(* Logix 5000 project; controller Hose_HP_Test_Rig_V1 vendor 1 type 14 code 149 rev 32.11; software revision 32.00; part 7 of 10 *)
(* tags used below, declared in another part *)
   GOTO_FAIL_BIN_STN1 : DINT;
   GOTO_FAULT_BIN_STN3 : DINT;
   PASS_COUNTER_STN1 : COUNTER;
   PASS_COUNTER_STN2 : COUNTER;
   PASS_COUNTER_STN3 : COUNTER;
   PASS_COUNTER_STN4 : COUNTER;
   ACT_PR_STN1 : REAL;
   ACT_PR_STN2 : REAL;
   ACT_PR_STN3 : REAL;
   ACT_PR_STN4 : REAL;
   AUTO_DOOR_OPEN_ON : BOOL;
   AUTO_DOOR_OPEN_ON_STN3 : BOOL;
   AUTO_TEST_ON_STN1 : BOOL;
   AUTO_TEST_ON_STN2 : BOOL;
   AUTO_TEST_ON_STN3 : BOOL;
   AUTO_TEST_ON_STN4 : BOOL;
   BOTTOM_CLAMP_AUTO_STN1 : BOOL;
   BOTTOM_CLAMP_AUTO_STN3 : BOOL;
   BOTTOM_CLAMP_C : REAL;
   BOTTOM_CLAMP_PR : REAL;
   BOTTOM_CLAMP_PR_SEL : BOOL;
   BOTTOM_CLAMP_PR_SEL_SET : BOOL;
   BOTTOM_CLAMP_PR_SEL_SOL : ALIAS FOR REM:O.Data[1].7;
   BOTTOM_CLAMP_SET_STN1 : BOOL;
   BOTTOM_CLAMP_SET_STN3 : BOOL;
   BOTTOM_CLAMP_SOL_STN1 : ALIAS FOR Local:1:O.Data.4;
   BOTTOM_CLAMP_SOL_STN3 : ALIAS FOR Local:3:O.Data.4;
   BOTTOM_CLAMP_X : REAL;
   BOTTOM_CLAMP_X1 : REAL;
   BOTTOM_CLAMP_X2 : REAL;
   BOTTOM_CLAMP_Y1 : REAL;
   BOTTOM_CLAMP_Y2 : REAL;
   BOTTOM_DECLAMP_AUTO_STN1 : BOOL;
   BOTTOM_DECLAMP_AUTO_STN3 : BOOL;
   BOTTOM_DECLAMP_SET_STN1 : BOOL;
   BOTTOM_DECLAMP_SET_STN3 : BOOL;
   BOTTOM_DECLAMP_SOL_STN1 : ALIAS FOR REM:O.Data[0].3;
   BOTTOM_DECLAMP_SOL_STN3 : ALIAS FOR REM:O.Data[0].7;
   BOTTOM_PR_SCL : SCP;
   BUZZER_STN1 : ALIAS FOR Local:3:O.Data.20;
   BUZZER_STN3 : ALIAS FOR Local:3:O.Data.29;
   CONS_FAIL_COUNT_STN1 : DINT;
   CONS_FAIL_COUNT_STN2 : DINT;
   CONS_FAIL_COUNT_STN3 : DINT;
   CONS_FAIL_COUNT_STN4 : DINT;
   CONS_FAIL_COUNTER_STN1 : COUNTER;
   CONS_FAIL_COUNTER_STN2 : COUNTER;
   CONS_FAIL_COUNTER_STN3 : COUNTER;
   CONS_FAIL_COUNTER_STN4 : COUNTER;
   CONSTRICTION_FILL_VAL_STN1 : BOOL;
   CONSTRICTION_FILL_VAL_STN3 : BOOL;
   CONSTRICTION_VALVE_SET_STN1 : BOOL;
   CONSTRICTION_VALVE_SET_STN3 : BOOL;
   DICH2_1_32 : DINT;
   DOOR_CLOSE_ABORT_STN1 : BOOL;
   DOOR_CLOSE_ABORT_STN3 : BOOL;
   DOOR_CLOSE_AUTO_STN1 : BOOL;
   DOOR_CLOSE_AUTO_STN3 : BOOL;
   DOOR_CLOSE_SET_STN1 : BOOL;
   DOOR_CLOSE_SET_STN3 : BOOL;
   DOOR_CLOSE_SOL_STN1 : ALIAS FOR Local:1:O.Data.2;
   DOOR_CLOSE_SOL_STN3 : ALIAS FOR Local:3:O.Data.2;
   DOOR_OPEN_SET_STN1 : BOOL;
   DOOR_OPEN_SET_STN3 : BOOL;
   DOOR_OPEN_SOL_STN1 : ALIAS FOR Local:1:O.Data.1;
   DOOR_OPEN_SOL_STN3 : ALIAS FOR Local:3:O.Data.1;
   EMG_FAULTED_STN1 : BOOL;
   EMG_FAULTED_STN3 : BOOL;
   EXHAUST_SET_STN1 : BOOL;
   EXHAUST_SET_STN3 : BOOL;
   EXHAUST_VALVE_STN1 : ALIAS FOR Local:1:O.Data.7;
   EXHAUST_VALVE_STN3 : ALIAS FOR Local:3:O.Data.7;
   EXHS_VAL_HP_ON_STN1 : BOOL;
   EXHS_VAL_HP_ON_STN3 : BOOL;
   EXHS_VAL_ON_STN1 : BOOL;
   EXHS_VAL_ON_STN3 : BOOL;
   FAIL_COUNT_RETEST : DINT;
   FAIL_COUNT_RETEST_STN2 : DINT;
   FAIL_COUNT_STN1 : DINT;
   FAIL_COUNT_STN2 : DINT;
   FAIL_COUNT_STN3 : DINT;
   FAIL_COUNT_STN4 : DINT;
   FAIL_COUNTER_RETEST : COUNTER;
   FAIL_COUNTER_RETEST_STN2 : COUNTER;
   FAIL_COUNTER_STN1 : COUNTER;
   FAIL_COUNTER_STN2 : COUNTER;
   FAIL_COUNTER_STN3 : COUNTER;
   FAIL_COUNTER_STN4 : COUNTER;
   FAILED_STN1 : BOOL;
   FAILED_STN3 : BOOL;
   FAULT_COUNT_STN1 : DINT;
   FAULT_COUNT_STN2 : DINT;
   FAULT_COUNT_STN3 : DINT;
   FAULT_COUNT_STN4 : DINT;
   FAULT_COUNTER_STN1 : COUNTER;
   FAULT_COUNTER_STN2 : COUNTER;
   FAULT_COUNTER_STN3 : COUNTER;
   FAULT_COUNTER_STN4 : COUNTER;
   FAULT_LAMP_STN1 : ALIAS FOR Local:3:O.Data.19;
   FAULT_LAMP_STN3 : ALIAS FOR Local:3:O.Data.28;
   FAULTED_STN1 : BOOL;
   FAULTED_STN3 : BOOL;
   FINAL_PR_BOTTOM_CLAMP : BOOL;
   FINAL_PR_STN1 : BOOL;
   FINAL_PR_STN2 : BOOL;
   FINAL_PR_STN3 : BOOL;
   FINAL_PR_STN4 : BOOL;
   FINAL_PR_TOP_CLAMP : BOOL;
   GOTO_FAIL_BIN_STN3 : DINT;
   GOTO_FAULT_BIN_STN1 : DINT;
   HIDE_MAIN_MENU : BOOL;
   HP_FILL_VALVE_SET_STN1 : BOOL;
   HP_FILL_VALVE_SET_STN3 : BOOL;
   HP_FILL_VALVE_STN1 : ALIAS FOR Local:1:O.Data.8;
   HP_FILL_VALVE_STN3 : ALIAS FOR Local:3:O.Data.8;
   INITIAL_PR_BOTTOM_CLAMP : BOOL;
   INITIAL_PR_STN1 : BOOL;
   INITIAL_PR_STN2 : BOOL;
   INITIAL_PR_STN3 : BOOL;
   INITIAL_PR_STN4 : BOOL;
   INITIAL_PR_TOP_CLAMP : BOOL;
   INPUT_1_16 : INT;
   MASTER_PR : REAL;
   MASTER_PR_CONS : REAL;
   MASTER_PR_SCL : SCP;
   MSB_EIP_1_16 : INT;
   PASS_COUNT_RETEST : DINT;
   PASS_COUNT_RETEST_STN2 : DINT;
   PASS_COUNT_STN1 : DINT;
   PASS_COUNT_STN2 : DINT;
   PASS_COUNT_STN3 : DINT;
   PASS_COUNT_STN4 : DINT;
   PASS_COUNTER_RETEST : COUNTER;
   PASS_COUNTER_RETEST_STN2 : COUNTER;
   PASS_LAMP_STN1 : ALIAS FOR Local:3:O.Data.18;
   PASS_LAMP_STN3 : ALIAS FOR Local:3:O.Data.27;
   PASSED_STN1 : BOOL;
   PASSED_STN3 : BOOL;
   PR_C_MASTER : REAL;
   PR_C_STAMP : REAL;
   PR_C_STN1 : REAL;
   PR_C_STN2 : REAL;
   PR_C_STN3 : REAL;
   PR_C_STN4 : REAL;
   PR_C_WORK : REAL;
   PR_DIFF_CALB_ACT : REAL;
   PR_SCL_STN1 : SCP;
   PR_SCL_STN2 : SCP;
   PR_SCL_STN3 : SCP;
   PR_SCL_STN4 : SCP;
   PR_X1_MASTER : REAL;
   PR_X1_STAMP : REAL;
   PR_X1_STN1 : REAL;
   PR_X1_STN2 : REAL;
   PR_X1_STN3 : REAL;
   PR_X1_STN4 : REAL;
   PR_X1_WORK : REAL;
   PR_X2_MASTER : REAL;
   PR_X2_STAMP : REAL;
   PR_X2_STN1 : REAL;
   PR_X2_STN2 : REAL;
   PR_X2_STN3 : REAL;
   PR_X2_STN4 : REAL;
   PR_X2_WORK : REAL;
   PR_X_MASTER : REAL;
   PR_X_STAMP : REAL;
   PR_X_STN1 : REAL;
   PR_X_STN2 : REAL;
   PR_X_STN3 : REAL;
   PR_X_STN4 : REAL;
   PR_X_WORK : REAL;
   PR_Y1_MASTER : REAL;
   PR_Y1_STAMP : REAL;
   PR_Y1_STN1 : REAL;
   PR_Y1_STN2 : REAL;
   PR_Y1_STN3 : REAL;
   PR_Y1_STN4 : REAL;
   PR_Y1_WORK : REAL;
   PR_Y2_MASTER : REAL;
   PR_Y2_STAMP : REAL;
   PR_Y2_STN1 : REAL;
   PR_Y2_STN2 : REAL;
   PR_Y2_STN3 : REAL;
   PR_Y2_STN4 : REAL;
   PR_Y2_WORK : REAL;
   RESET_COUNT_RETEST : BOOL;
   RESET_COUNT_RETEST_STN2 : BOOL;
   RESET_COUNT_STN1 : BOOL;
   RESET_COUNT_STN2 : BOOL;
   RESET_COUNT_STN3 : BOOL;
   RESET_COUNT_STN4 : BOOL;
   RST_BOTTOM_DECLAMP_STN1 : BOOL;
   RST_BOTTOM_DECLAMP_STN3 : BOOL;
   RST_DOOR_OPEN_ON : BOOL;
   RST_DOOR_OPEN_ON_STN3 : BOOL;
   RST_TOP_DECLAMP_AUTO_STN1 : BOOL;
   RST_TOP_DECLAMP_AUTO_STN3 : BOOL;
   STAMP_ON_STN1 : BOOL;
   STAMP_ON_STN3 : BOOL;
   STAMP_PR : REAL;
   STAMP_PR_SCL : SCP;
   STAMP_SOL_STN1 : ALIAS FOR Local:1:O.Data.5;
   STAMP_SOL_STN3 : ALIAS FOR Local:3:O.Data.5;
   STS : DINT;
   TEST_LAMP_STN1 : ALIAS FOR Local:3:O.Data.17;
   TEST_LAMP_STN3 : ALIAS FOR Local:3:O.Data.26;
   TEST_SOL_STN1 : ALIAS FOR Local:1:O.Data.6;
   TEST_SOL_STN3 : ALIAS FOR Local:3:O.Data.6;
   TEST_VAL_ON_STN1 : BOOL;
   TEST_VAL_ON_STN3 : BOOL;
   TOP_CLAMP_AUTO_STN1 : BOOL;
   TOP_CLAMP_AUTO_STN3 : BOOL;
   TOP_CLAMP_C : REAL;
   TOP_CLAMP_PR : REAL;
   TOP_CLAMP_PR_SEL : BOOL;
   TOP_CLAMP_PR_SEL_SET : BOOL;
   TOP_CLAMP_PR_SEL_SOL : ALIAS FOR REM:O.Data[1].6;
   TOP_CLAMP_SET_STN1 : BOOL;
   TOP_CLAMP_SET_STN3 : BOOL;
   TOP_CLAMP_SOL_STN1 : ALIAS FOR Local:1:O.Data.3;
   TOP_CLAMP_SOL_STN3 : ALIAS FOR Local:3:O.Data.3;
   TOP_CLAMP_X : REAL;
   TOP_CLAMP_X1 : REAL;
   TOP_CLAMP_X2 : REAL;
   TOP_CLAMP_Y1 : REAL;
   TOP_CLAMP_Y2 : REAL;
   TOP_DECLAMP_AUTO_STN1 : BOOL;
   TOP_DECLAMP_AUTO_STN3 : BOOL;
   TOP_DECLAMP_SET_STN1 : BOOL;
   TOP_DECLAMP_SET_STN3 : BOOL;
   TOP_DECLAMP_SOL_STN1 : ALIAS FOR REM:O.Data[0].2;
   TOP_DECLAMP_SOL_STN3 : ALIAS FOR REM:O.Data[0].6;
   TOP_PR_SCL : SCP;
   TOTAL_PASS_COUNT : DINT;
   WORK_PR_CONS : REAL;
   WORK_PR_PT : REAL;
   WORK_PR_SCL : SCP;
(* MainProgram, continued *)

ROUTINE MainRoutine   (* ladder *)
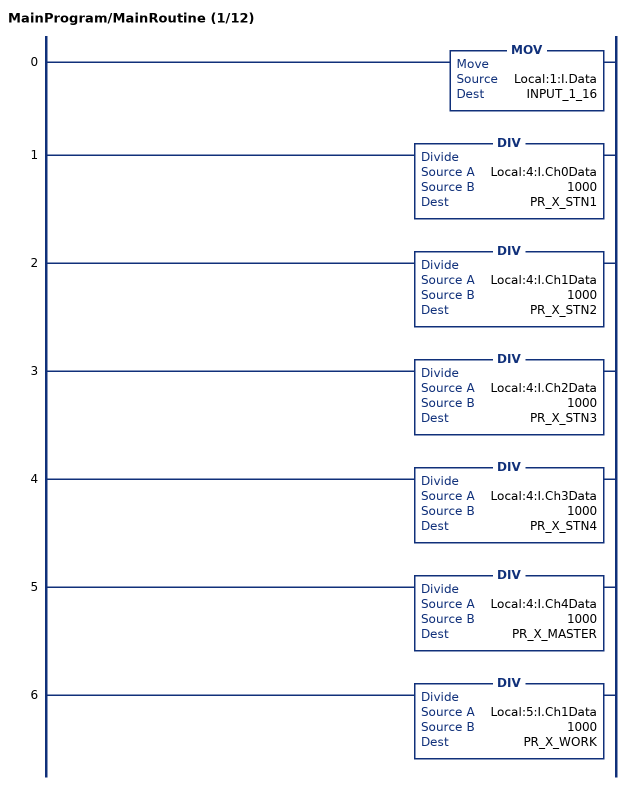
   0: MOV(Local:1:I.Data,INPUT_1_16);
   1: DIV(Local:4:I.Ch0Data,1000,PR_X_STN1);
   2: DIV(Local:4:I.Ch1Data,1000,PR_X_STN2);
   3: DIV(Local:4:I.Ch2Data,1000,PR_X_STN3);
   4: DIV(Local:4:I.Ch3Data,1000,PR_X_STN4);
   5: DIV(Local:4:I.Ch4Data,1000,PR_X_MASTER);
   6: DIV(Local:5:I.Ch1Data,1000,PR_X_WORK);
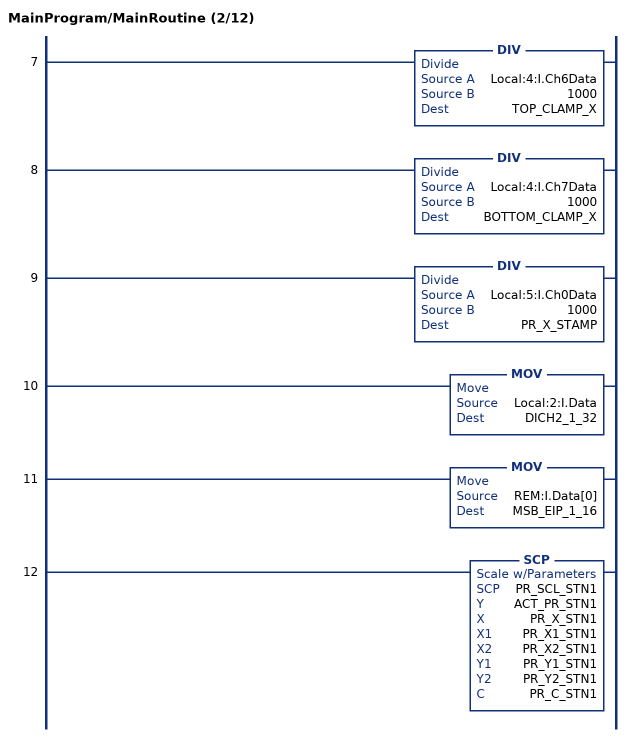
   7: DIV(Local:4:I.Ch6Data,1000,TOP_CLAMP_X);
   8: DIV(Local:4:I.Ch7Data,1000,BOTTOM_CLAMP_X);
   9: DIV(Local:5:I.Ch0Data,1000,PR_X_STAMP);
   10: MOV(Local:2:I.Data,DICH2_1_32);
   11: MOV(REM:I.Data[0],MSB_EIP_1_16);
   12: SCP(PR_SCL_STN1,ACT_PR_STN1,PR_X_STN1,PR_X1_STN1,PR_X2_STN1,PR_Y1_STN1,PR_Y2_STN1,PR_C_STN1);
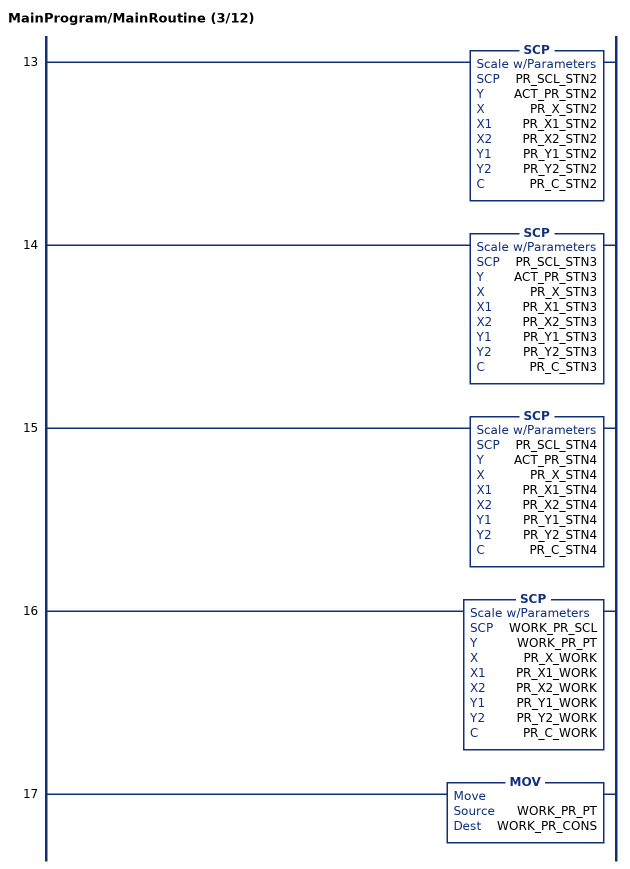
   13: SCP(PR_SCL_STN2,ACT_PR_STN2,PR_X_STN2,PR_X1_STN2,PR_X2_STN2,PR_Y1_STN2,PR_Y2_STN2,PR_C_STN2);
   14: SCP(PR_SCL_STN3,ACT_PR_STN3,PR_X_STN3,PR_X1_STN3,PR_X2_STN3,PR_Y1_STN3,PR_Y2_STN3,PR_C_STN3);
   15: SCP(PR_SCL_STN4,ACT_PR_STN4,PR_X_STN4,PR_X1_STN4,PR_X2_STN4,PR_Y1_STN4,PR_Y2_STN4,PR_C_STN4);
   16: SCP(WORK_PR_SCL,WORK_PR_PT,PR_X_WORK,PR_X1_WORK,PR_X2_WORK,PR_Y1_WORK,PR_Y2_WORK,PR_C_WORK);
   17: MOV(WORK_PR_PT,WORK_PR_CONS);
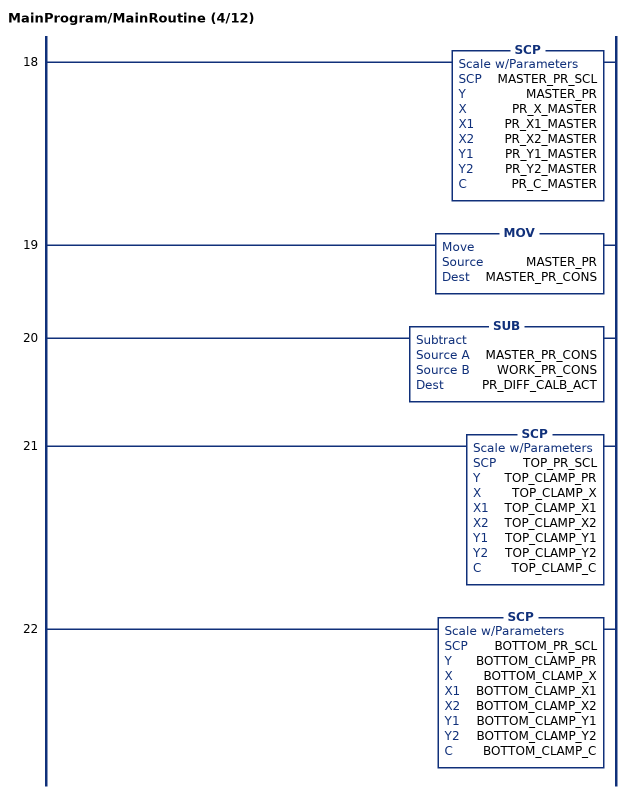
   18: SCP(MASTER_PR_SCL,MASTER_PR,PR_X_MASTER,PR_X1_MASTER,PR_X2_MASTER,PR_Y1_MASTER,PR_Y2_MASTER,PR_C_MASTER);
   19: MOV(MASTER_PR,MASTER_PR_CONS);
   20: SUB(MASTER_PR_CONS,WORK_PR_CONS,PR_DIFF_CALB_ACT);
   21: SCP(TOP_PR_SCL,TOP_CLAMP_PR,TOP_CLAMP_X,TOP_CLAMP_X1,TOP_CLAMP_X2,TOP_CLAMP_Y1,TOP_CLAMP_Y2,TOP_CLAMP_C);
   22: SCP(BOTTOM_PR_SCL,BOTTOM_CLAMP_PR,BOTTOM_CLAMP_X,BOTTOM_CLAMP_X1,BOTTOM_CLAMP_X2,BOTTOM_CLAMP_Y1,BOTTOM_CLAMP_Y2,BOTTOM_CLAMP_C);
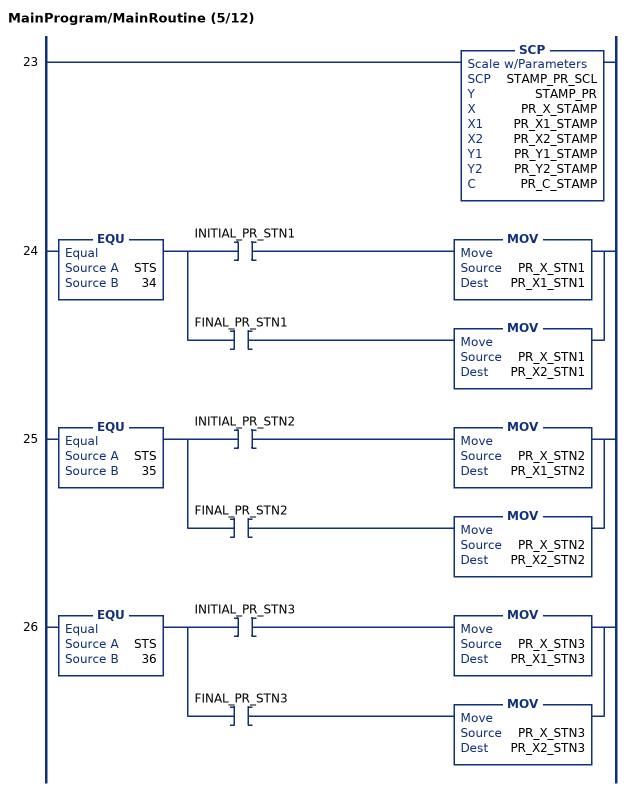
   23: SCP(STAMP_PR_SCL,STAMP_PR,PR_X_STAMP,PR_X1_STAMP,PR_X2_STAMP,PR_Y1_STAMP,PR_Y2_STAMP,PR_C_STAMP);
   24: EQU(STS,34)[XIC(INITIAL_PR_STN1) MOV(PR_X_STN1,PR_X1_STN1) ,XIC(FINAL_PR_STN1) MOV(PR_X_STN1,PR_X2_STN1) ];
   25: EQU(STS,35)[XIC(INITIAL_PR_STN2) MOV(PR_X_STN2,PR_X1_STN2) ,XIC(FINAL_PR_STN2) MOV(PR_X_STN2,PR_X2_STN2) ];
   26: EQU(STS,36)[XIC(INITIAL_PR_STN3) MOV(PR_X_STN3,PR_X1_STN3) ,XIC(FINAL_PR_STN3) MOV(PR_X_STN3,PR_X2_STN3) ];
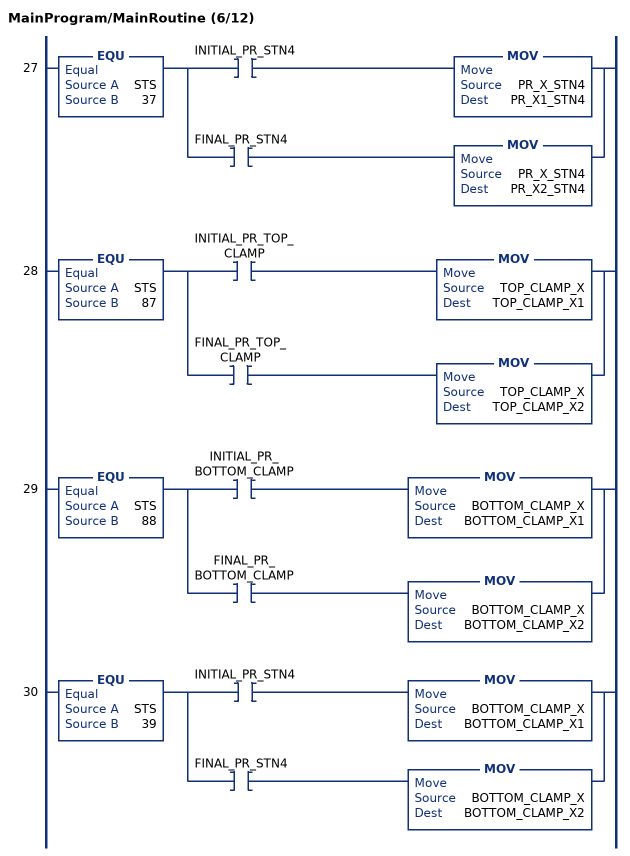
   27: EQU(STS,37)[XIC(INITIAL_PR_STN4) MOV(PR_X_STN4,PR_X1_STN4) ,XIC(FINAL_PR_STN4) MOV(PR_X_STN4,PR_X2_STN4) ];
   28: EQU(STS,87)[XIC(INITIAL_PR_TOP_CLAMP) MOV(TOP_CLAMP_X,TOP_CLAMP_X1) ,XIC(FINAL_PR_TOP_CLAMP) MOV(TOP_CLAMP_X,TOP_CLAMP_X2) ];
   29: EQU(STS,88)[XIC(INITIAL_PR_BOTTOM_CLAMP) MOV(BOTTOM_CLAMP_X,BOTTOM_CLAMP_X1) ,XIC(FINAL_PR_BOTTOM_CLAMP) MOV(BOTTOM_CLAMP_X,BOTTOM_CLAMP_X2) ];
   30: EQU(STS,39)[XIC(INITIAL_PR_STN4) MOV(BOTTOM_CLAMP_X,BOTTOM_CLAMP_X1) ,XIC(FINAL_PR_STN4) MOV(BOTTOM_CLAMP_X,BOTTOM_CLAMP_X2) ];
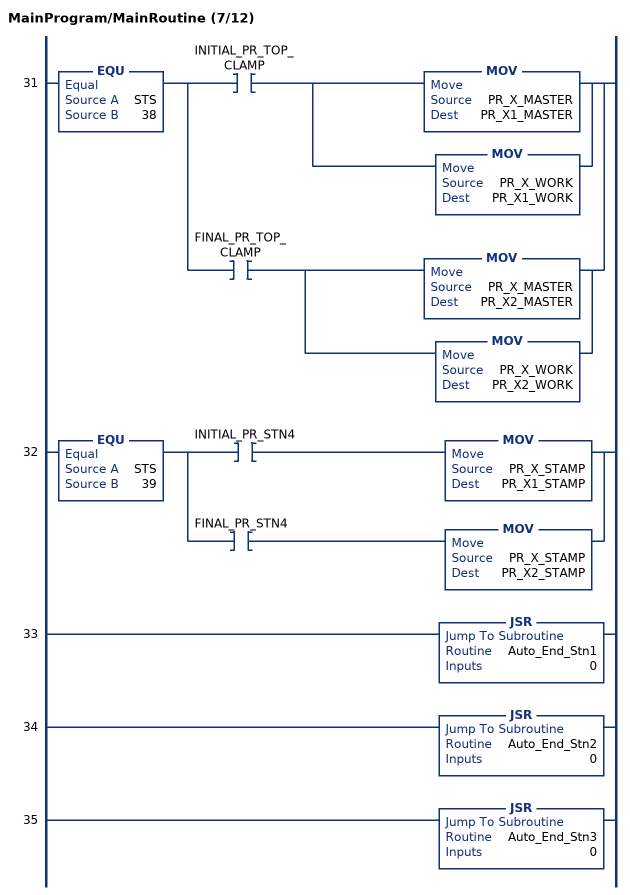
   31: EQU(STS,38)[XIC(INITIAL_PR_TOP_CLAMP) [MOV(PR_X_MASTER,PR_X1_MASTER) ,MOV(PR_X_WORK,PR_X1_WORK) ] ,XIC(FINAL_PR_TOP_CLAMP) [MOV(PR_X_MASTER,PR_X2_MASTER) ,MOV(PR_X_WORK,PR_X2_WORK) ] ];
   32: EQU(STS,39)[XIC(INITIAL_PR_STN4) MOV(PR_X_STAMP,PR_X1_STAMP) ,XIC(FINAL_PR_STN4) MOV(PR_X_STAMP,PR_X2_STAMP) ];
   33: JSR(Auto_End_Stn1,0);
   34: JSR(Auto_End_Stn2,0);
   35: JSR(Auto_End_Stn3,0);
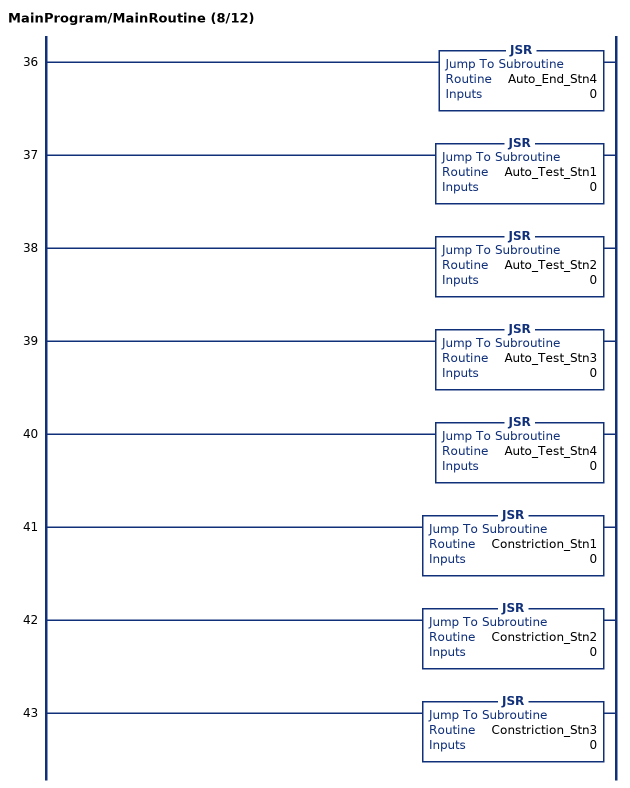
   36: JSR(Auto_End_Stn4,0);
   37: JSR(Auto_Test_Stn1,0);
   38: JSR(Auto_Test_Stn2,0);
   39: JSR(Auto_Test_Stn3,0);
   40: JSR(Auto_Test_Stn4,0);
   41: JSR(Constriction_Stn1,0);
   42: JSR(Constriction_Stn2,0);
   43: JSR(Constriction_Stn3,0);
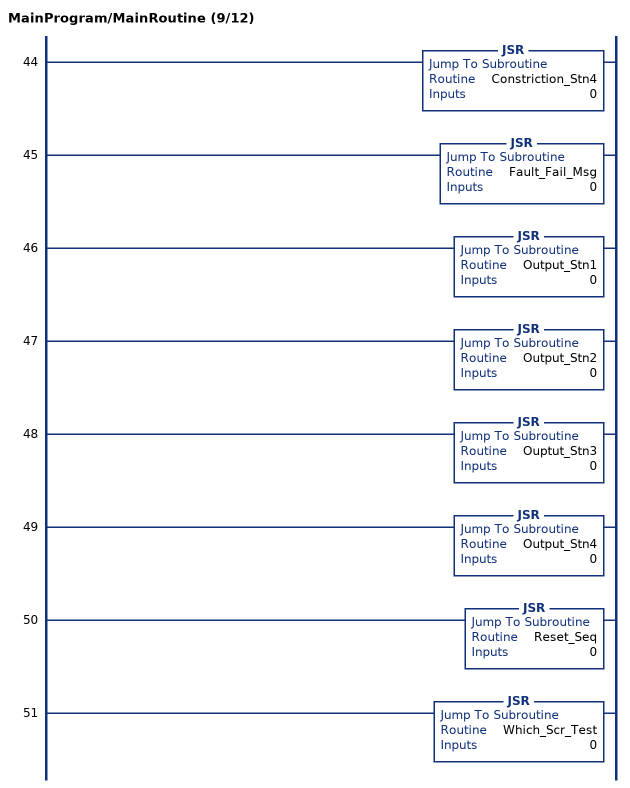
   44: JSR(Constriction_Stn4,0);
   45: JSR(Fault_Fail_Msg,0);
   46: JSR(Output_Stn1,0);
   47: JSR(Output_Stn2,0);
   48: JSR(Ouptut_Stn3,0);
   49: JSR(Output_Stn4,0);
   50: JSR(Reset_Seq,0);
   51: JSR(Which_Scr_Test,0);
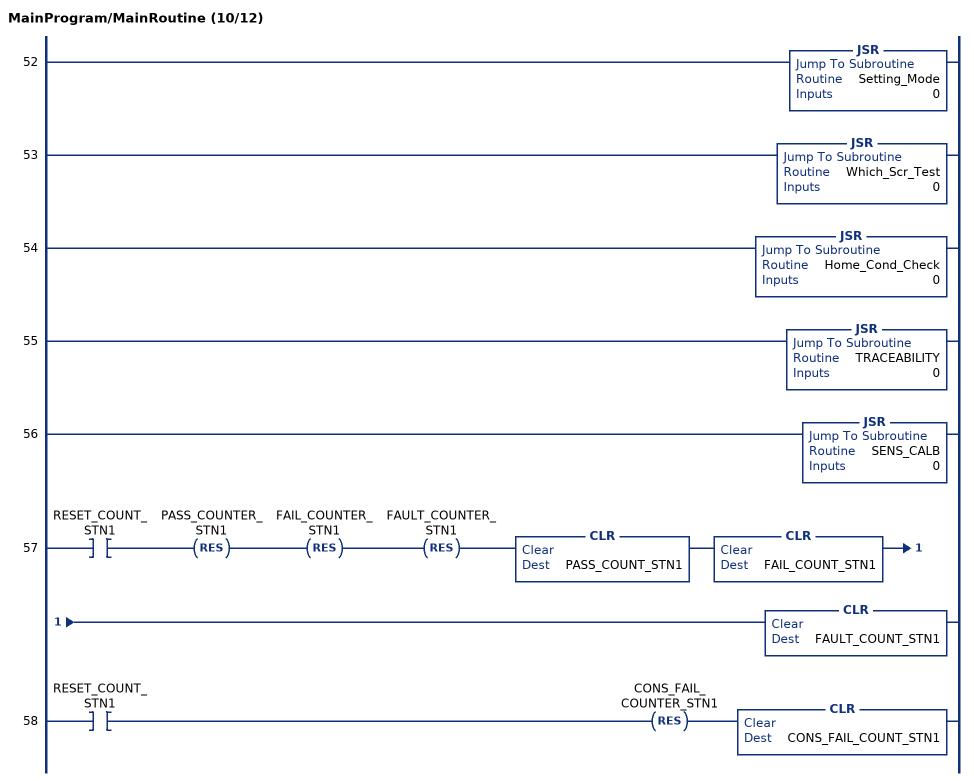
   52: JSR(Setting_Mode,0);
   53: JSR(Which_Scr_Test,0);
   54: JSR(Home_Cond_Check,0);
   55: JSR(TRACEABILITY,0);
   56: JSR(SENS_CALB,0);
   57: XIC(RESET_COUNT_STN1)RES(PASS_COUNTER_STN1)RES(FAIL_COUNTER_STN1)RES(FAULT_COUNTER_STN1)CLR(PASS_COUNT_STN1)CLR(FAIL_COUNT_STN1)CLR(FAULT_COUNT_STN1);
   58: XIC(RESET_COUNT_STN1)RES(CONS_FAIL_COUNTER_STN1)CLR(CONS_FAIL_COUNT_STN1);
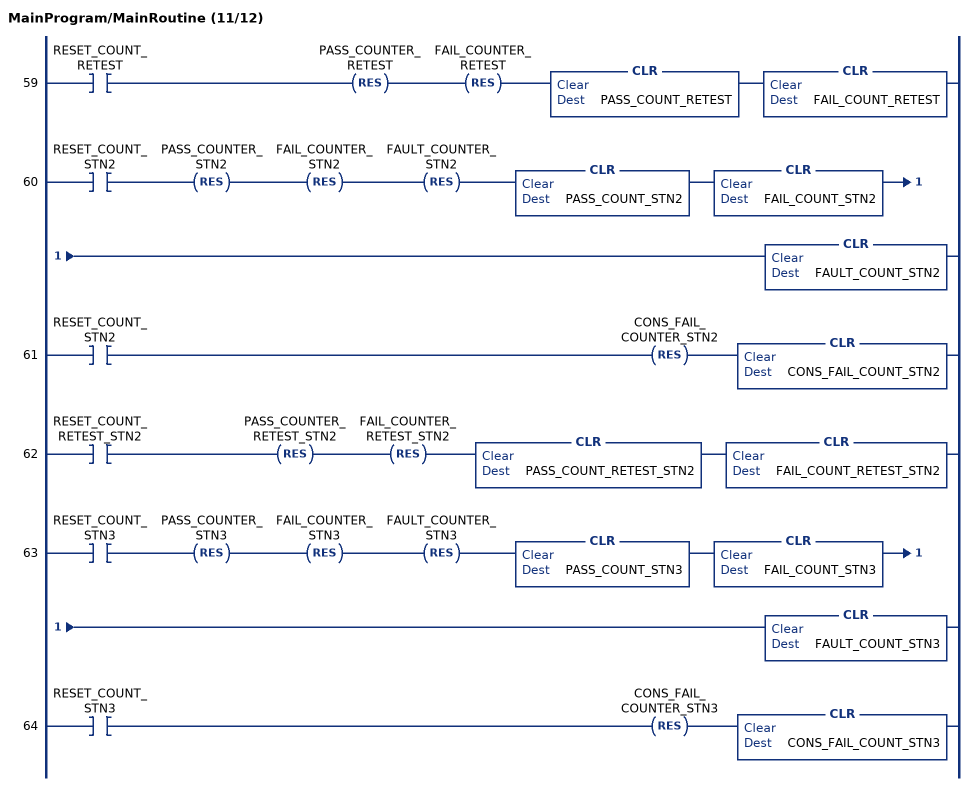
   59: XIC(RESET_COUNT_RETEST)RES(PASS_COUNTER_RETEST)RES(FAIL_COUNTER_RETEST)CLR(PASS_COUNT_RETEST)CLR(FAIL_COUNT_RETEST);
   60: XIC(RESET_COUNT_STN2)RES(PASS_COUNTER_STN2)RES(FAIL_COUNTER_STN2)RES(FAULT_COUNTER_STN2)CLR(PASS_COUNT_STN2)CLR(FAIL_COUNT_STN2)CLR(FAULT_COUNT_STN2);
   61: XIC(RESET_COUNT_STN2)RES(CONS_FAIL_COUNTER_STN2)CLR(CONS_FAIL_COUNT_STN2);
   62: XIC(RESET_COUNT_RETEST_STN2)RES(PASS_COUNTER_RETEST_STN2)RES(FAIL_COUNTER_RETEST_STN2)CLR(PASS_COUNT_RETEST_STN2)CLR(FAIL_COUNT_RETEST_STN2);
   63: XIC(RESET_COUNT_STN3)RES(PASS_COUNTER_STN3)RES(FAIL_COUNTER_STN3)RES(FAULT_COUNTER_STN3)CLR(PASS_COUNT_STN3)CLR(FAIL_COUNT_STN3)CLR(FAULT_COUNT_STN3);
   64: XIC(RESET_COUNT_STN3)RES(CONS_FAIL_COUNTER_STN3)CLR(CONS_FAIL_COUNT_STN3);
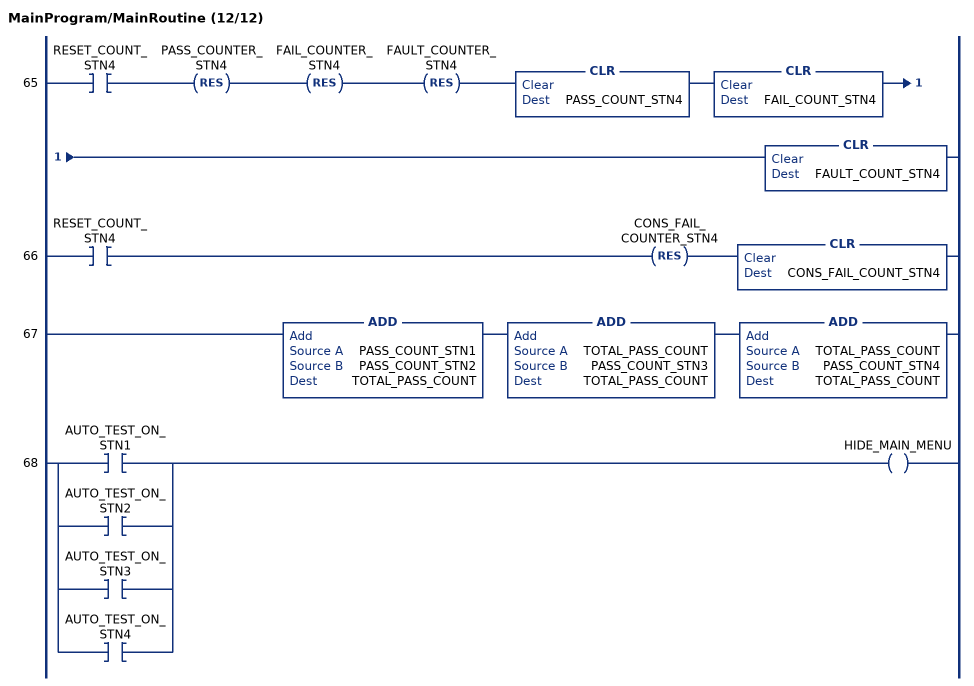
   65: XIC(RESET_COUNT_STN4)RES(PASS_COUNTER_STN4)RES(FAIL_COUNTER_STN4)RES(FAULT_COUNTER_STN4)CLR(PASS_COUNT_STN4)CLR(FAIL_COUNT_STN4)CLR(FAULT_COUNT_STN4);
   66: XIC(RESET_COUNT_STN4)RES(CONS_FAIL_COUNTER_STN4)CLR(CONS_FAIL_COUNT_STN4);
   67: ADD(PASS_COUNT_STN1,PASS_COUNT_STN2,TOTAL_PASS_COUNT)ADD(TOTAL_PASS_COUNT,PASS_COUNT_STN3,TOTAL_PASS_COUNT)ADD(TOTAL_PASS_COUNT,PASS_COUNT_STN4,TOTAL_PASS_COUNT);
   68: [XIC(AUTO_TEST_ON_STN1) ,XIC(AUTO_TEST_ON_STN2) ,XIC(AUTO_TEST_ON_STN3) ,XIC(AUTO_TEST_ON_STN4) ]OTE(HIDE_MAIN_MENU);
END_ROUTINE

ROUTINE Ouptut_Stn3   (* ladder *)
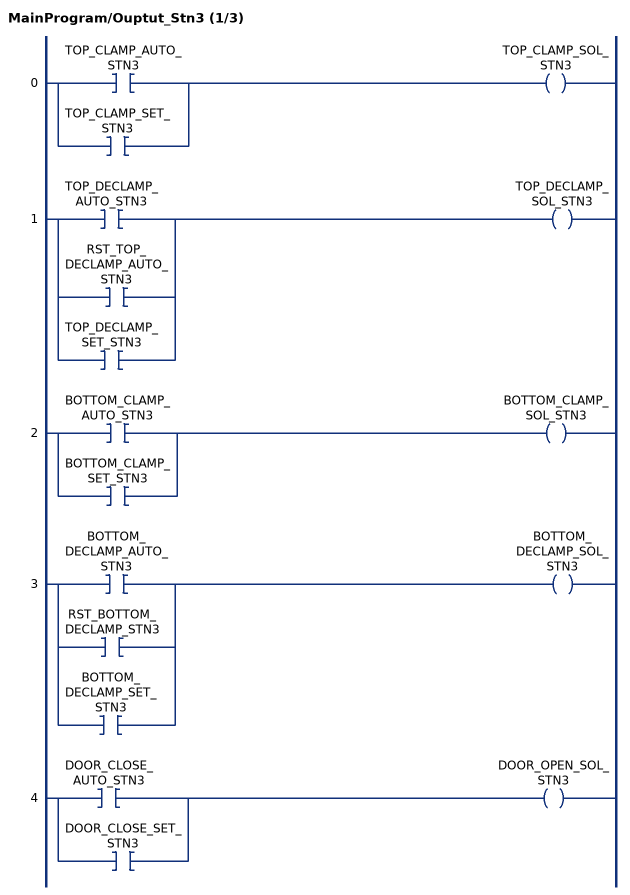
   0: [XIC(TOP_CLAMP_AUTO_STN3) ,XIC(TOP_CLAMP_SET_STN3) ]OTE(TOP_CLAMP_SOL_STN3);
   1: [XIC(TOP_DECLAMP_AUTO_STN3) ,XIC(RST_TOP_DECLAMP_AUTO_STN3) ,XIC(TOP_DECLAMP_SET_STN3) ]OTE(TOP_DECLAMP_SOL_STN3);
   2: [XIC(BOTTOM_CLAMP_AUTO_STN3) ,XIC(BOTTOM_CLAMP_SET_STN3) ]OTE(BOTTOM_CLAMP_SOL_STN3);
   3: [XIC(BOTTOM_DECLAMP_AUTO_STN3) ,XIC(RST_BOTTOM_DECLAMP_STN3) ,XIC(BOTTOM_DECLAMP_SET_STN3) ]OTE(BOTTOM_DECLAMP_SOL_STN3);
   4: [XIC(DOOR_CLOSE_AUTO_STN3) ,XIC(DOOR_CLOSE_SET_STN3) ]OTE(DOOR_OPEN_SOL_STN3);
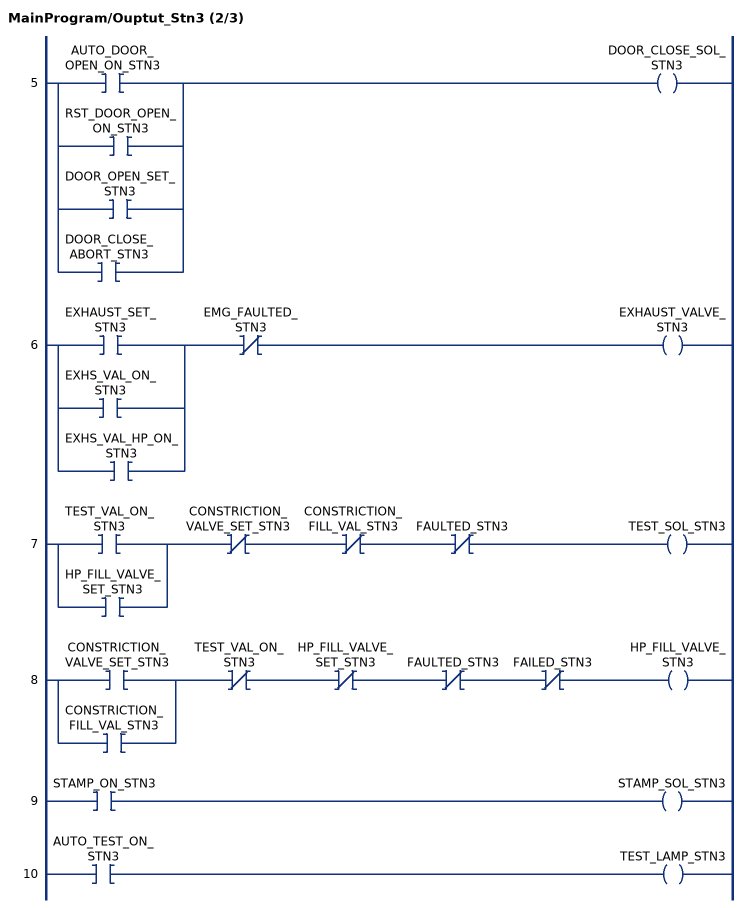
   5: [XIC(AUTO_DOOR_OPEN_ON_STN3) ,XIC(RST_DOOR_OPEN_ON_STN3) ,XIC(DOOR_OPEN_SET_STN3) ,XIC(DOOR_CLOSE_ABORT_STN3) ]OTE(DOOR_CLOSE_SOL_STN3);
   6: [XIC(EXHAUST_SET_STN3) ,XIC(EXHS_VAL_ON_STN3) ,XIC(EXHS_VAL_HP_ON_STN3) ]XIO(EMG_FAULTED_STN3)OTE(EXHAUST_VALVE_STN3);
   7: [XIC(TEST_VAL_ON_STN3) ,XIC(HP_FILL_VALVE_SET_STN3) ]XIO(CONSTRICTION_VALVE_SET_STN3)XIO(CONSTRICTION_FILL_VAL_STN3)XIO(FAULTED_STN3)OTE(TEST_SOL_STN3);
   8: [XIC(CONSTRICTION_VALVE_SET_STN3) ,XIC(CONSTRICTION_FILL_VAL_STN3) ]XIO(TEST_VAL_ON_STN3)XIO(HP_FILL_VALVE_SET_STN3)XIO(FAULTED_STN3)XIO(FAILED_STN3)OTE(HP_FILL_VALVE_STN3);
   9: XIC(STAMP_ON_STN3)OTE(STAMP_SOL_STN3);
   10: XIC(AUTO_TEST_ON_STN3)OTE(TEST_LAMP_STN3);
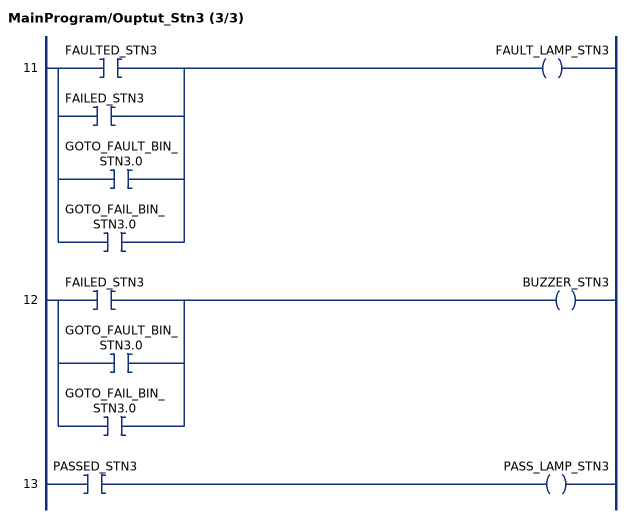
   11: [XIC(FAULTED_STN3) ,XIC(FAILED_STN3) ,XIC(GOTO_FAULT_BIN_STN3.0) ,XIC(GOTO_FAIL_BIN_STN3.0) ]OTE(FAULT_LAMP_STN3);
   12: [XIC(FAILED_STN3) ,XIC(GOTO_FAULT_BIN_STN3.0) ,XIC(GOTO_FAIL_BIN_STN3.0) ]OTE(BUZZER_STN3);
   13: XIC(PASSED_STN3)OTE(PASS_LAMP_STN3);
END_ROUTINE

ROUTINE Output_Stn1   (* ladder *)
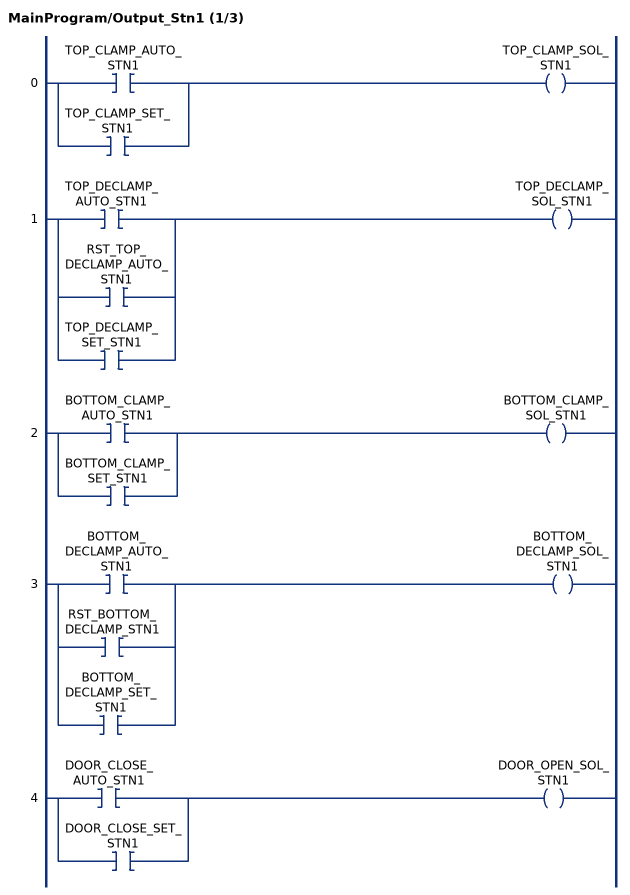
   0: [XIC(TOP_CLAMP_AUTO_STN1) ,XIC(TOP_CLAMP_SET_STN1) ]OTE(TOP_CLAMP_SOL_STN1);
   1: [XIC(TOP_DECLAMP_AUTO_STN1) ,XIC(RST_TOP_DECLAMP_AUTO_STN1) ,XIC(TOP_DECLAMP_SET_STN1) ]OTE(TOP_DECLAMP_SOL_STN1);
   2: [XIC(BOTTOM_CLAMP_AUTO_STN1) ,XIC(BOTTOM_CLAMP_SET_STN1) ]OTE(BOTTOM_CLAMP_SOL_STN1);
   3: [XIC(BOTTOM_DECLAMP_AUTO_STN1) ,XIC(RST_BOTTOM_DECLAMP_STN1) ,XIC(BOTTOM_DECLAMP_SET_STN1) ]OTE(BOTTOM_DECLAMP_SOL_STN1);
   4: [XIC(DOOR_CLOSE_AUTO_STN1) ,XIC(DOOR_CLOSE_SET_STN1) ]OTE(DOOR_OPEN_SOL_STN1);
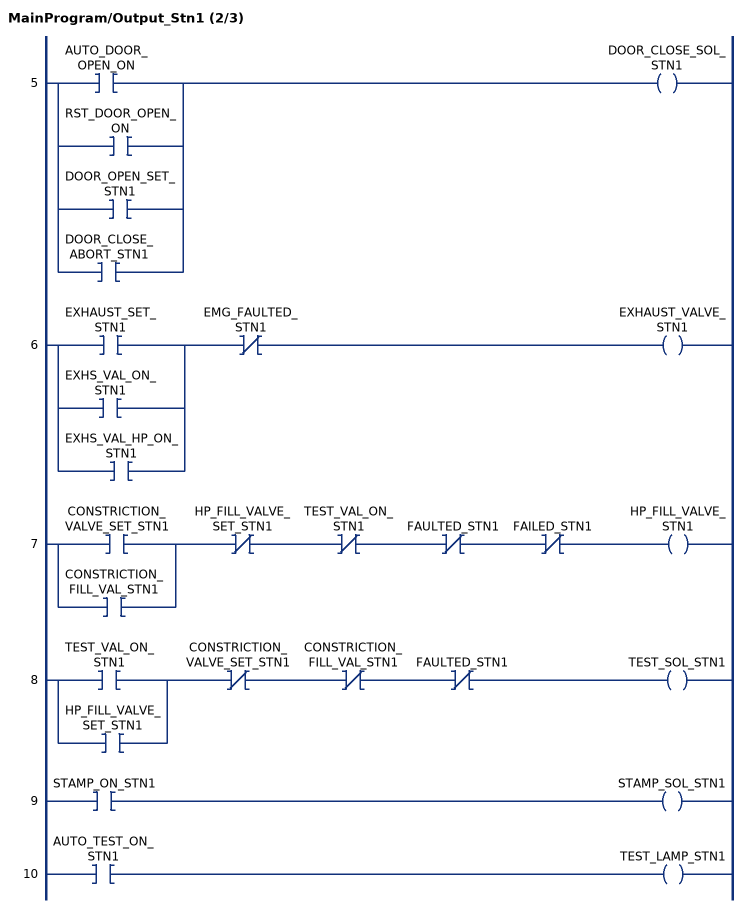
   5: [XIC(AUTO_DOOR_OPEN_ON) ,XIC(RST_DOOR_OPEN_ON) ,XIC(DOOR_OPEN_SET_STN1) ,XIC(DOOR_CLOSE_ABORT_STN1) ]OTE(DOOR_CLOSE_SOL_STN1);
   6: [XIC(EXHAUST_SET_STN1) ,XIC(EXHS_VAL_ON_STN1) ,XIC(EXHS_VAL_HP_ON_STN1) ]XIO(EMG_FAULTED_STN1)OTE(EXHAUST_VALVE_STN1);
   7: [XIC(CONSTRICTION_VALVE_SET_STN1) ,XIC(CONSTRICTION_FILL_VAL_STN1) ]XIO(HP_FILL_VALVE_SET_STN1)XIO(TEST_VAL_ON_STN1)XIO(FAULTED_STN1)XIO(FAILED_STN1)OTE(HP_FILL_VALVE_STN1);
   8: [XIC(TEST_VAL_ON_STN1) ,XIC(HP_FILL_VALVE_SET_STN1) ]XIO(CONSTRICTION_VALVE_SET_STN1)XIO(CONSTRICTION_FILL_VAL_STN1)XIO(FAULTED_STN1)OTE(TEST_SOL_STN1);
   9: XIC(STAMP_ON_STN1)OTE(STAMP_SOL_STN1);
   10: XIC(AUTO_TEST_ON_STN1)OTE(TEST_LAMP_STN1);
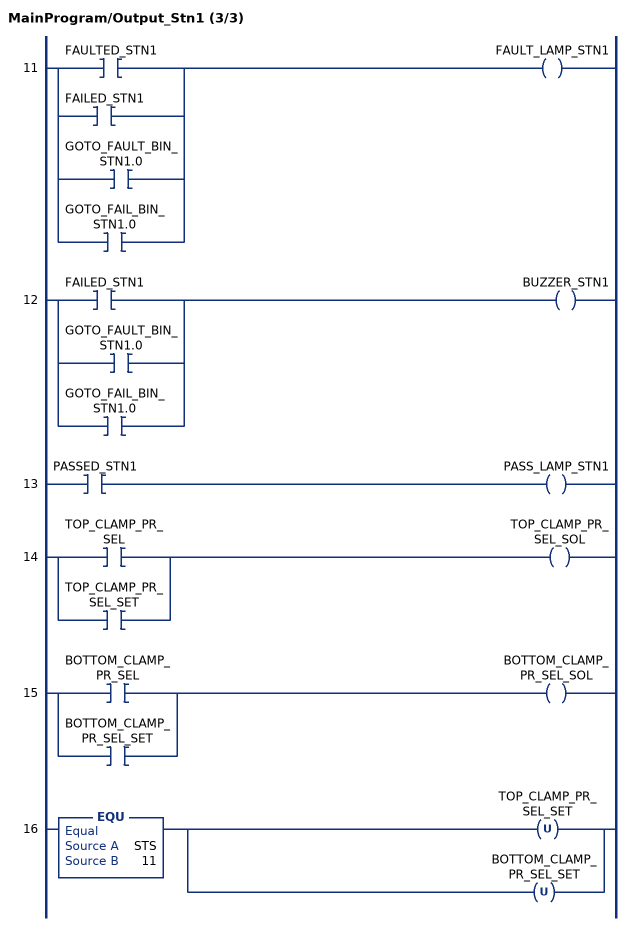
   11: [XIC(FAULTED_STN1) ,XIC(FAILED_STN1) ,XIC(GOTO_FAULT_BIN_STN1.0) ,XIC(GOTO_FAIL_BIN_STN1.0) ]OTE(FAULT_LAMP_STN1);
   12: [XIC(FAILED_STN1) ,XIC(GOTO_FAULT_BIN_STN1.0) ,XIC(GOTO_FAIL_BIN_STN1.0) ]OTE(BUZZER_STN1);
   13: XIC(PASSED_STN1)OTE(PASS_LAMP_STN1);
   14: [XIC(TOP_CLAMP_PR_SEL) ,XIC(TOP_CLAMP_PR_SEL_SET) ]OTE(TOP_CLAMP_PR_SEL_SOL);
   15: [XIC(BOTTOM_CLAMP_PR_SEL) ,XIC(BOTTOM_CLAMP_PR_SEL_SET) ]OTE(BOTTOM_CLAMP_PR_SEL_SOL);
   16: EQU(STS,11)[OTU(TOP_CLAMP_PR_SEL_SET) ,OTU(BOTTOM_CLAMP_PR_SEL_SET) ];
END_ROUTINE
